// TIA Portal V19 export
DATA_BLOCK "DB_SNTP_Diag"   // DB202
{ S7_Optimized_Access := 'TRUE' }
// stored: AutoNumber false, MemoryReserve 100
   VAR
      error : Bool;   // An error occured
      statusID : Int;   // Specifies the source of the error (1 = TCON, 2 = TUSEND, 3 = TURCV)
      status : Word;   // Specifies the error
      lastStatusID : Int;   // Saved status ID
      lastStatus : Word;   // Saved status
   END_VAR
BEGIN
END_DATA_BLOCK
